(* PLC project device, CODESYS STW CODESYS V3.5 SP11 - ESX-3CS *)
(* stored: creationDateTime 2026-05-19T11:33:34.046707, version 0.1, modificationDateTime 2026-01-26T16:59:03, organization Isoloader *)

TYPE t_persistent_bool : PersistentBool;
END_TYPE

TYPE t_persistent_DWORD : PersistentDWORD;
END_TYPE

TYPE t_persistent_int : PersistentINT;
END_TYPE

TYPE t_persistent_medium_string : PersistentMediumString;
END_TYPE

TYPE t_persistent_real : PersistentReal;
END_TYPE

TYPE t_persistent_short_string : PersistentShortString;
END_TYPE

TYPE t_persistent_store : PersistentStore;
END_TYPE

TYPE t_persistent_uint : PersistentUINT;
END_TYPE

TYPE t_persistent_ULINT : PersistentULINT;
END_TYPE

TYPE t_store_buffer : ARRAY[0..cStoreBufferSize] OF BYTE;
END_TYPE

TYPE t_store_type : STRUCT
  buffer : t_store_buffer;
  enabled : BOOL;
END_STRUCT;
END_TYPE

VAR_GLOBAL CONSTANT  (* GlobalVariablesDevice *)
  cStoreBufferSize : UINT := 2798;
  gPersistenceManager : PersistenceManager;
END_VAR

FUNCTION_BLOCK HeartbeatHandler EXTENDS ReceiveCANMessage
  VAR
    lHeartbeatTimer : t_timer;
  END_VAR

            
          

METHOD initialize
                  SUPER^.initialize();

lHeartbeatTimer.Period := T#300MS;
lHeartbeatTimer.Enable := TRUE;
lHeartbeatTimer.initialize();


                
END_METHOD

METHOD operator
                  SUPER^.operator();

lHeartbeatTimer.operator();

IF (Received) THEN
	lHeartbeatTimer.reset();
END_IF

                
END_METHOD

METHOD initializeMessage
  VAR_INPUT
    handle : UDINT;
    channel : USINT;
  END_VAR
                  lHandler.ou32_Handle := handle;


                
END_METHOD

PROPERTY Period : t_time
GET
                    Period := lHeartbeatTimer.Period;
                  
END_GET
SET
                    lHeartbeatTimer.Period := Period;
                  
END_SET
END_PROPERTY

PROPERTY HeartbeatFault : BOOL
GET
                    HeartbeatFault := lHeartbeatTimer.Expired;
                  
END_GET
END_PROPERTY
END_FUNCTION_BLOCK

FUNCTION_BLOCK ReceiveCANMessage EXTENDS CANMessage
  VAR
    lHandle : UDINT;
    lHandler : FB_x_can_obj_get_msg;
    lMessage : T_x_can_msg;
    lReturnStatus : INT;
    lReceived : BOOL;
    lReceivedCount : UINT := 0;
    lTimer : t_timer;
    lProceedOnFail : BOOL := TRUE;
    lProceedOnTimeout : BOOL := TRUE;
  END_VAR

            
          

METHOD initializeReceive
  VAR_INPUT
    handle : UDINT;
  END_VAR
                  ;
                
END_METHOD

METHOD operator
                  SUPER^.operator();

lHandler(ou32_Handle := lHandle,ot_Msg => lMessage,os16_Status => lReturnStatus);

IF (lReturnStatus=C_NO_ERR) THEN
	lReceivedCount := lReceivedCount + 1;

	lReceived := TRUE;
	lSuccess := TRUE;
	lFinished := TRUE;
	lProceed := TRUE;
	
	finish();
	RETURN;
END_IF

IF (lReturnStatus<>C_NOACT) THEN
	lReceived := FALSE;
	lSuccess := FALSE;
	lFinished := TRUE;
	lProceed := lProceedOnFail;
	
	finish();
	RETURN;	
END_IF

lTimer.operator();
IF (lTimer.Expired) THEN
	lReceived := FALSE;
	lSuccess := FALSE;
	lFinished := TRUE;
	lProceed := lProceedOnTimeout;
	
	finish();
	RETURN;	
END_IF

lReceived := FALSE;

                
END_METHOD

METHOD reset
                  lReceived := FALSE;
                
END_METHOD

METHOD start
                  SUPER^.start();

lTImer.reset();
                
END_METHOD

METHOD initialize
                  SUPER^.initialize();

lReceivedCount := 0;

lTimer.Enable := TRUE;
lTimer.Period := T#1S;
lTimer.initialize();
                
END_METHOD

PROPERTY Handle : UDINT
GET
                    Handle := lHandle;
                  
END_GET
SET
                    lHandle := Handle;
                  
END_SET
END_PROPERTY

PROPERTY Period : t_time
GET
                    Period := lTImer.Period;
                  
END_GET
SET
                    lTimer.Period := Period;
                  
END_SET
END_PROPERTY

PROPERTY Received : BOOL
GET
                    Received := lReceived;
                  
END_GET
END_PROPERTY
END_FUNCTION_BLOCK

FUNCTION_BLOCK SDOReadCANMessage EXTENDS CANMessage
  VAR
    lSDORead : CIA405.SDO_READ_DATA;
    lSDOReadData : DWORD;
    lSDODReadDataLength : UDINT;
    lSDOReadAttemptCounter : USINT := 0;  (* lSDOLastSuccessfulReadData: DWORD; *)
    lSDOReadSuccessCounter : USINT := 0;
    lProceedOnFail : BOOL := TRUE;
    lProceedOnOverflow : BOOL := TRUE;
  END_VAR

            
          

METHOD cancelSDORead
                  lSDORead.ENABLE := FALSE;
lSDORead(DATALENGTH:=lSDODReadDataLength);

                
END_METHOD

METHOD initialize
                  SUPER^.initialize();

lSDOReadAttemptCounter := 0;
lSDOReadSuccessCounter := 0;

lSDORead.CHANNEL := 0;
lSDORead.ENABLE := FALSE;
lSDORead.TIMEOUT := 500;
lSDORead.MODE := CIA405.SDO_MODE.AUTO;
lSDORead.DATA := ADR(lSDOReadData);
                
END_METHOD

METHOD operator
                  SUPER^.operator();

IF (lSDORead.ENABLE) THEN
	lSDORead(DATALENGTH:=lSDODReadDataLength);
	IF ((lSDORead.CONFIRM) OR (lSDORead.ERROR<>CIA405.CANOPEN_KERNEL_ERROR.CANOPEN_KERNEL_NO_ERROR)) THEN
		lSDORead.ENABLE := FALSE;
		lSDOReadAttemptCounter := lSDOReadAttemptCounter + 1;
		IF (lSDORead.CONFIRM) THEN
			lSuccess := TRUE;
			lFinished := TRUE;
			lProceed := TRUE;
			
			sdoReadHandler();
			lSDOReadSuccessCounter := lSDOReadSuccessCounter + 1;
			
			finish();
			RETURN;
		END_IF
		IF (lSDORead.ERROR<>CIA405.CANOPEN_KERNEL_ERROR.CANOPEN_KERNEL_NO_ERROR) THEN
			lSuccess := FALSE;
			lFinished := TRUE;
			lProceed := TRUE;
			
			finish();
			RETURN;
		END_IF
	END_IF	
END_IF

                
END_METHOD

METHOD reset
                  SUPER^.reset();
                
END_METHOD

METHOD sdoReadHandler
                  ;
                
END_METHOD

METHOD start
                  cancelSDORead();
lSDORead.ENABLE := TRUE;

SUPER^.start();
                
END_METHOD
END_FUNCTION_BLOCK

FUNCTION_BLOCK SDOWriteCANMessage EXTENDS CANMessage
  VAR
    lSDOWrite : CIA405.SDO_WRITE_DATA;
    lSDOWriteData : DWORD;
    lSDOWriteAttemptCounter : USINT := 0;
    lSDOWriteSuccessCounter : USINT := 0;
    lProceedOnFail : BOOL := TRUE;
    lProceedOnOverflow : BOOL := TRUE;
  END_VAR

            
          

METHOD cancelSDOWrite
                  lSDOWrite.ENABLE := FALSE;
lSDOWrite();
                
END_METHOD

METHOD initialize
                  SUPER^.initialize();

lSDOWriteAttemptCounter := 0;
lSDOWriteSuccessCounter := 0;

lSDOWrite.CHANNEL := 0;
lSDOWrite.ENABLE := FALSE;
lSDOWrite.TIMEOUT := 500;
lSDOWrite.MODE := CIA405.SDO_MODE.AUTO;
lSDOWrite.DATA := ADR(lSDOWriteData);
                
END_METHOD

METHOD operator
                  SUPER^.operator();

IF (lSDOWrite.ENABLE) THEN
	lSDOWrite();
	IF ((lSDOWrite.CONFIRM) OR (lSDOWrite.ERROR<>CIA405.CANOPEN_KERNEL_ERROR.CANOPEN_KERNEL_NO_ERROR)) THEN
		lSDOWrite.ENABLE := FALSE;
		lSDOWriteAttemptCounter := lSDOWriteAttemptCounter + 1;
		IF (lSDOWrite.CONFIRM) THEN
			lSuccess := TRUE;
			lFinished := TRUE;
			lProceed := TRUE;
			
			lSDOWriteSuccessCounter := lSDOWriteSuccessCounter + 1;
			
			finish();
			RETURN;
		END_IF
		IF (lSDOWrite.ERROR<>CIA405.CANOPEN_KERNEL_ERROR.CANOPEN_KERNEL_NO_ERROR) THEN
			lSuccess := FALSE;
			lFinished := TRUE;
			lProceed := TRUE;
			
			finish();
			RETURN;
		END_IF
	END_IF	
END_IF


                
END_METHOD

METHOD reset
                  SUPER^.reset();
                
END_METHOD

METHOD start
                  cancelSDOWrite();
lSDOWrite.ENABLE := TRUE;

SUPER^.start();
                
END_METHOD
END_FUNCTION_BLOCK

FUNCTION_BLOCK TransmitCANMessage EXTENDS CANMessage
  VAR
    lHandle : UDINT;
    lHandler : FB_x_can_obj_send_msg;
    lMessage : T_x_can_msg;
    lReturnStatus : INT;
    lTransmitted : BOOL;
    lTransmittedCount : UINT := 0;
    lProceedOnFail : BOOL := TRUE;
    lProceedOnOverflow : BOOL := TRUE;
  END_VAR

            
          

METHOD initialize
  VAR_INPUT
    handle : UDINT;
  END_VAR
                  SUPER^.initialize();

lTransmittedCount := 0;
                
END_METHOD

METHOD operator
                  SUPER^.operator();

lHandler(lHandle,lMessage,lReturnStatus);

IF (lReturnStatus=C_NO_ERR) THEN
	lTransmittedCount := lTransmittedCount + 1;

	lTransmitted := TRUE;
	lSuccess := TRUE;
	lFinished := TRUE;
	lProceed := TRUE;
	
	finish();
	RETURN;
END_IF

IF (lReturnStatus<>C_OVERFLOW) THEN
	lTransmitted := FALSE;
	lSuccess := FALSE;
	lFinished := TRUE;
	lProceed := lProceedOnFail;
	
	finish();
	RETURN;	
END_IF

lTransmitted := FALSE;
lSuccess := FALSE;
lFinished := TRUE;
lProceed := lProceedOnOverflow;

finish();

                
END_METHOD

METHOD reset
                  lTransmitted := false;
                
END_METHOD

METHOD start
                  SUPER^.start();

                
END_METHOD
END_FUNCTION_BLOCK

FUNCTION_BLOCK TransmitMessage
  VAR
    lHandler : FB_x_can_obj_send_msg;
    lMessage : T_x_can_msg;
    lReturnStatus : INT;
    lOverflowCount : UINT := 0;
  END_VAR

            
          

METHOD initializeMessage
  VAR_INPUT
    handle : UDINT;
    channel : USINT;
  END_VAR
                  lHandler.ou32_Handle := handle;


                
END_METHOD

METHOD initialize
                  reset();

                
END_METHOD

METHOD operator
                  lHandler(ot_Msg := lMessage,os16_Status => lReturnStatus);

IF (lReturnStatus=C_OVERFLOW) THEN
	lOverflowCount := lOverflowCount + 1;
END_IF
                
END_METHOD

METHOD reset
                  lOverflowCount := 0;
                
END_METHOD

METHOD transmit : INT
  VAR_INPUT
    message : T_x_can_msg;
  END_VAR
                  lHandler(ot_Msg := message,os16_Status => lReturnStatus);

IF (lReturnStatus=C_OVERFLOW) THEN
	lOverflowCount := lOverflowCount + 1;
END_IF

transmit := lReturnStatus;
                
END_METHOD
END_FUNCTION_BLOCK

FUNCTION_BLOCK TransmitNMT EXTENDS TransmitMessage

            
          

METHOD initialize
                  SUPER^.initialize();

lMessage.t_Id.u32_Id := 16#0;
lMessage.t_Id.u8_Xtd := X_OFF;
lMessage.u8_Dlc := 2;
lMessage.au8_Data[0] := 0;
lMessage.au8_Data[1] := 0;

                
END_METHOD

METHOD preOperationalAllNodes
                  lMessage.au8_Data[0] := 128;
lMessage.au8_Data[1] := 0;

operator();
                
END_METHOD

METHOD preOperationalNode
  VAR_INPUT
    node : USINT;
  END_VAR
                  lMessage.au8_Data[0] := 128;
lMessage.au8_Data[1] := node;

operator();
                
END_METHOD

METHOD resetAllNodes
                  lMessage.au8_Data[0] := 129;
lMessage.au8_Data[1] := 0;

operator();
                
END_METHOD

METHOD resetNode
  VAR_INPUT
    node : USINT;
  END_VAR
                  lMessage.au8_Data[0] := 129;
lMessage.au8_Data[1] := node;

operator();
                
END_METHOD

METHOD startAllNodes
                  lMessage.au8_Data[0] := 1;
lMessage.au8_Data[1] := 0;

operator();
                
END_METHOD

METHOD startNode
  VAR_INPUT
    node : USINT;
  END_VAR
                  lMessage.au8_Data[0] := 1;
lMessage.au8_Data[1] := node;

operator();
                
END_METHOD

METHOD stopAllNodes
                  lMessage.au8_Data[0] := 2;
lMessage.au8_Data[1] := 0;

operator();
                
END_METHOD

METHOD stopNode
  VAR_INPUT
    node : USINT;
  END_VAR
                  lMessage.au8_Data[0] := 2;
lMessage.au8_Data[1] := node;

operator();
                
END_METHOD
END_FUNCTION_BLOCK

FUNCTION_BLOCK TransmitSDO EXTENDS TransmitMessage

            
          

METHOD initialize
                  SUPER^.initialize();

lMessage.t_Id.u32_Id := 16#0;
lMessage.t_Id.u8_Xtd := X_OFF;
lMessage.u8_Dlc := 2;
lMessage.au8_Data[0] := 0;
lMessage.au8_Data[1] := 0;

                
END_METHOD

METHOD stopAllNodes
                  lMessage.au8_Data[0] := 2;
lMessage.au8_Data[1] := 0;

operator();
                
END_METHOD

METHOD stopNode
  VAR_INPUT
    node : USINT;
  END_VAR
                  lMessage.au8_Data[0] := 2;
lMessage.au8_Data[1] := node;

operator();
                
END_METHOD
END_FUNCTION_BLOCK

FUNCTION_BLOCK PersistenceManager
  VAR CONSTANT
    cBlockSize : USINT := 4;
    cAllocatedBlockMax : UDINT := 6101;
  END_VAR
  VAR
    lAllocated : UDINT := 0;
    lWriteCounter : UDINT := 0;
  END_VAR

            
          

METHOD allocate : UDINT
  VAR_INPUT
    sz : UDINT;
    id : t_persistent_id;
    blocks : REFERENCE TO UINT;
  END_VAR
  VAR
    address : UDINT;
  END_VAR
                  allocate := INT_TO_UINT(id) * cBlockSize;

blocks := REAL_TO_UINT(UDINT_TO_REAL(sz)/USINT_TO_REAL(cBlockSize));
IF ((blocks*cBlockSize)<sz) THEN
	blocks := blocks + 1;
END_IF

lAllocated := MAX(allocate + sz,lAllocated);

IF (lAllocated>(cAllocatedBlockMax*cBlockSize)) THEN
	gCodeErrorHandler(pMessage:='over allocation in PersistenceManager');
END_IF
                
END_METHOD

METHOD clear
  VAR
    lData : ARRAY[0..cAllocatedBlockMax] OF DWORD;
    lHandler : FB_x_eep_write;
    i : UDINT;
  END_VAR
                  FOR i:=0 TO cAllocatedBlockMax DO
	lData[i] := 0;
END_FOR

lHandler.ou32_Address := 0;
lHandler.ou32_Count := SIZEOF(lData);
lHandler.opu8_Data := ADR(lData);

lHandler();

                
END_METHOD

METHOD read : DWORD
  VAR_INPUT
    index : UDINT;
  END_VAR
  VAR
    lHandler : FB_x_eep_read;
    data : DWORD;
  END_VAR
                  lHandler.ou32_Address := MIN(index,cAllocatedBlockMax)*cBlockSize;
lHandler.ou32_Count := cBlockSize;
lHandler.opu8_Data := ADR(data);

lHandler();
read := data;

                
END_METHOD

METHOD write
  VAR_INPUT
    index : UDINT;
    data : DWORD;
  END_VAR
  VAR
    lHandler : FB_x_eep_write;
    lFlush : FB_x_eep_flush;
  END_VAR
                  lHandler.ou32_Address := MIN(index,cAllocatedBlockMax)*cBlockSize;
lHandler.ou32_Count := cBlockSize;
lHandler.opu8_Data := ADR(data);

lHandler();
lFlush();
                
END_METHOD

PROPERTY WriteCounter : UDINT
GET
                    WriteCounter := lWriteCounter;
                  
END_GET
SET
                    lWriteCounter := WriteCounter + 1;
                  
END_SET
END_PROPERTY

PROPERTY IndexMax : UDINT
GET
                    IndexMax := lAllocated/cBlockSize;
                  
END_GET
END_PROPERTY
END_FUNCTION_BLOCK

FUNCTION_BLOCK PersistentBool EXTENDS PersistentValue
  VAR
    lValue : BOOL;
  END_VAR

            
          

METHOD initialize
                  lData := ADR(lValue);
lCount := SIZEOF(lValue);

SUPER^.initialize();
                
END_METHOD

PROPERTY Value : BOOL
GET
                    Value := lValue;
                  
END_GET
SET
                    IF (Value=lValue) THEN
	RETURN;
END_IF

lValue := Value;
write();



                  
END_SET
END_PROPERTY
END_FUNCTION_BLOCK

FUNCTION_BLOCK PersistentDWORD EXTENDS PersistentValue
  VAR
    lValue : DWORD;
  END_VAR

            
          

METHOD initialize
                  lData := ADR(lValue);
lCount := SIZEOF(lValue);

SUPER^.initialize();

IF (lValue=NOT(16#0)) THEN //foobar why?
	lValue := 16#0;
END_IF

                
END_METHOD

PROPERTY Value : DWORD
GET
                    Value := lValue;
                  
END_GET
SET
                    IF (Value=lValue) THEN
	RETURN;
END_IF

lValue := Value;
write();
                  
END_SET
END_PROPERTY
END_FUNCTION_BLOCK

FUNCTION_BLOCK PersistentINT EXTENDS PersistentValue
  VAR
    lValue : INT;
  END_VAR

            
          

METHOD initialize
                  lData := ADR(lValue);
lCount := SIZEOF(lValue);

SUPER^.initialize();
                
END_METHOD

PROPERTY Value : INT
GET
                    Value := lValue;
                  
END_GET
SET
                    IF (Value=lValue) THEN
	RETURN;
END_IF

lValue := Value;
write();



                  
END_SET
END_PROPERTY
END_FUNCTION_BLOCK

FUNCTION_BLOCK PersistentMediumString EXTENDS PersistentValue
  VAR
    lValue : t_medium_string;
  END_VAR

            
          

METHOD initialize
                  lData := ADR(lValue[0]);
lCount := SIZEOF(lValue);

SUPER^.initialize();


                
END_METHOD

PROPERTY Value : t_medium_string
GET
                    IF (lValue[0]=255) THEN
	Value := '';
	RETURN;
END_IF

Value := lValue;

                  
END_GET
SET
                    IF (strcmp(Value,lValue)) THEN
	RETURN;
END_IF

lValue := Value;
write();
                  
END_SET
END_PROPERTY
END_FUNCTION_BLOCK

FUNCTION_BLOCK PersistentReal EXTENDS PersistentValue
  VAR
    lValue : REAL;
  END_VAR

            
          

METHOD initialize
                  lData := ADR(lValue);
lCount := SIZEOF(lValue);

SUPER^.initialize();

                
END_METHOD

(* {attribute 'monitoring' := 'call'} *)
PROPERTY Value : REAL
GET
                    Value := lValue;
                  
END_GET
SET
                    IF (Value=lValue) THEN
	RETURN;
END_IF

lValue := Value;
write();
                  
END_SET
END_PROPERTY
END_FUNCTION_BLOCK

FUNCTION_BLOCK PersistentShortString EXTENDS PersistentValue
  VAR
    lValue : t_short_string;
  END_VAR

            
          

METHOD initialize
                  lData := ADR(lValue[0]);
lCount := SIZEOF(lValue);

SUPER^.initialize();

                
END_METHOD

PROPERTY Value : t_short_string
GET
                    IF (lValue[0]=255) THEN
	Value := '';
	RETURN;
END_IF

Value := lValue;
                  
END_GET
SET
                    IF (strcmp(Value,lValue)) THEN
	RETURN;
END_IF

lValue := Value;
write();

                  
END_SET
END_PROPERTY
END_FUNCTION_BLOCK

FUNCTION_BLOCK PersistentStore EXTENDS PersistentValue
  VAR
    lValue : t_store_type;
  END_VAR

            
          

METHOD initialize
                  lData := ADR(lValue);
lCount := SIZEOF(lValue);

SUPER^.initialize();


                
END_METHOD

METHOD clear
                  MEMUtils.MemSet(ADR(lValue),0,UDINT_TO_DWORD(lCount));
write();

                
END_METHOD

METHOD export
  VAR_INPUT
    store : REFERENCE TO t_store_type;
  END_VAR
                  IF (NOT(__ISVALIDREF(store))) THEN
	RETURN;	
END_IF

MEMUtils.MemCpy(ADR(store),ADR(lValue),UDINT_TO_DWORD(lCount));

                
END_METHOD

METHOD import
  VAR_INPUT
    store : REFERENCE TO t_store_type;
  END_VAR
                  IF (NOT(__ISVALIDREF(store))) THEN
	RETURN;	
END_IF

IF (MEMUtils.MemCmp(ADR(lValue),ADR(store),UDINT_TO_DWORD(lCount))) THEN
	RETURN;
END_IF

MEMUtils.MemCpy(ADR(lValue),ADR(store),UDINT_TO_DWORD(lCount));
write();
                
END_METHOD
END_FUNCTION_BLOCK

FUNCTION_BLOCK PersistentUINT EXTENDS PersistentValue
  VAR
    lValue : UINT;
  END_VAR

            
          

METHOD initialize
                  lData := ADR(lValue);
lCount := SIZEOF(lValue);

SUPER^.initialize();
                
END_METHOD

PROPERTY Value : UINT
GET
                    Value := lValue;
                  
END_GET
SET
                    IF (Value=lValue) THEN
	RETURN;
END_IF

lValue := Value;
write();



                  
END_SET
END_PROPERTY
END_FUNCTION_BLOCK

FUNCTION_BLOCK PersistentULINT EXTENDS PersistentValue
  VAR
    lValue : ULINT;
  END_VAR

            
          

METHOD initialize
                  lData := ADR(lValue);
lCount := SIZEOF(lValue);

SUPER^.initialize();
                
END_METHOD

PROPERTY Value : ULINT
GET
                    Value := lValue;
                  
END_GET
SET
                    IF (Value=lValue) THEN
	RETURN;
END_IF

lValue := Value;
write();



                  
END_SET
END_PROPERTY
END_FUNCTION_BLOCK

FUNCTION_BLOCK PersistentValue
  VAR
    lReadHandler : FB_x_eep_read;
    lWriteHandler : FB_x_eep_write;
    lIdentifier : t_persistent_id := t_persistent_id.cPersistentID_Default;
    lAddress : UDINT := 0;
    lCount : UDINT := 0;
    lBlocks : UINT := 0;
    lData : POINTER TO USINT := 0;
    lWriteCounter : UINT := 0;
  END_VAR

            
          

METHOD initialize
                  lAddress := gPersistenceManager.allocate(lCount,lIdentifier,lBlocks);

lReadHandler.ou32_Address := lAddress;
lReadHandler.ou32_Count := lCount;
lReadHandler.opu8_Data := lData;

lWriteHandler.ou32_Address := lAddress;
lWriteHandler.ou32_Count := lCount;
lWriteHandler.opu8_Data := lData;

read();
                
END_METHOD

METHOD read
                  lReadHandler();
                
END_METHOD

METHOD write
                  lWriteHandler();

lWriteCounter := lWriteCounter + 1;
gPersistenceManager.WriteCounter := gPersistenceManager.WriteCounter + 1;

                
END_METHOD

PROPERTY Identifier : t_persistent_id
GET
                    Identifier := lIdentifier;
                  
END_GET
SET
                    lIdentifier := Identifier;
                  
END_SET
END_PROPERTY

PROPERTY Blocks : UINT
GET
                    Blocks := lBlocks;
                  
END_GET
END_PROPERTY
END_FUNCTION_BLOCK

FUNCTION fIsValidTCPHandle : BOOL
  VAR_INPUT
    handle : RTS_IEC_HANDLE;
  END_VAR

            fIsValidTCPHandle := (handle<>CmpErrors.SysTypes.RTS_INVALID_HANDLE);

          
END_FUNCTION
